// TIA Portal V19 export
TYPE "LEXCHANGETRAY_typeAxisSimpleControlProcessValues_2"
// stored: Access Published
   STRUCT
      enable : Bool;
      referenceDesignator : String[154];
      enabled : Bool;
      enableManualCmds : Bool;
      enableAxis : Bool;
      axisEnabled : Bool;
      resetAxis : Bool;
      home : Bool;
      halt : Bool;
      posAbsolute : Bool;
      posRelative : Bool;
      moveVelocity : Bool;
      jogForward : Bool;
      jogBackward : Bool;
      stop : Bool;
      enableTorque : Bool;
      readValues : Bool;
      resetDone : Bool;
      resetBusy : Bool;
      resetAborted : Bool;
      homeDone : Bool;
      homeBusy : Bool;
      homeAborted : Bool;
      haltDone : Bool;
      haltBusy : Bool;
      haltAborted : Bool;
      posAbsoluteDone : Bool;
      posAbsoluteBusy : Bool;
      posAbsoluteAborted : Bool;
      posRelativeDone : Bool;
      posRelativeBusy : Bool;
      posRelativeAborted : Bool;
      inVelocity : Bool;
      moveVelocityBusy : Bool;
      moveVolocityAborted : Bool;
      jogInVelocity : Bool;
      jogBusy : Bool;
      jogAborted : Bool;
      torqueBusy : Bool;
      InClamping : Bool;
      InLimitation : Bool;
      stopDone : Bool;
      stopBusy : Bool;
      stopAborted : Bool;
      valid : Bool;
      busy : Bool;
      error : Bool;
      status : Word;
      subfunctionStatus : Word;
      axisType : UDInt;
      statusWord : "LBC_typeAxisSimpleControlStatusWord";
      warningWord { S7_SetPoint := 'True'} : "LBC_typeAxisSimpleControlWarningWord";
      errorWord { S7_SetPoint := 'True'} : "LBC_typeAxisSimpleControlErrorWord";
      errorNumber { S7_SetPoint := 'True'} : UDInt;
      errorReaction : DInt;
      position : LReal;
      velocity : LReal;
      actualPosition : LReal;
      actualVelocity : LReal;
      actualTorque : LReal;
      targetPosition : LReal;
      followingError : LReal;
      lengthUnit : UDInt;
      velocityUnit : UDInt;
   END_STRUCT;
END_TYPE
